(* CODESYS project TIMER.project

Project tree, tasks and I/O mapping:
  Device : CODESYS Control Win V3, 3S - Smart Software Solutions GmbH, order no. 305021, version 3.5.11.30
    application Application
      libraries: Standard, * (System)
      task MainTask (cyclic, interval t#20ms, priority 1) calls PLC_PRG
      program PLC_PRG [LD]
*)

// Device/Application/PLC_PRG
PROGRAM PLC_PRG
VAR
	START : BOOL;               // INICIA O SISTEMA
	STOP : BOOL;                // PARA O SISTEMA
	SISTEMA: BOOL;              // FUNCIONAMENTO
	S1 : BOOL;                  // SENSOR DETECTOR DE GARRAFAS
	P1: BOOL;
	P2: BOOL;
	VS : BOOL;                  // VALVULA SOLENOIDE
	TON_1: TON;
	T1: TIME;
	P3: BOOL;
END_VAR

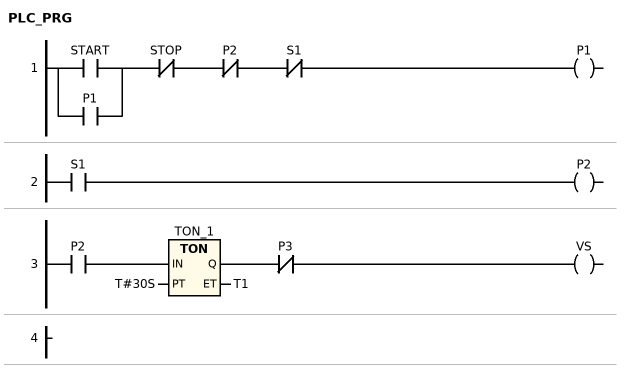
// NETWORK 1
P1 := (START OR P1) AND NOT STOP AND NOT P2 AND NOT S1;

// NETWORK 2
P2 := S1;

// NETWORK 3
TON_1(IN := P2, PT := T#30S, ET => T1); // TON
VS := TON_1.Q AND NOT P3;

// NETWORK 4

END_PROGRAM
